FUNCTION_BLOCK PUBLIC FB_BANNER_K50
VAR_IN_OUT
	Hardware : TYP_BAN_K50_HW;
END_VAR
VAR_INPUT
END_VAR
VAR_OUTPUT
	ButtonPressed : BOOL;
	ButtonPosEdge : BOOL;
	ButtonNegEdge : BOOL;
END_VAR
VAR
	PosTrig : R_TRIG;
	NegTrig : F_TRIG;
END_VAR

ButtonPressed := Hardware.In.ButtonPressed;

PosTrig(CLK := ButtonPressed, Q => ButtonPosEdge);
NegTrig(CLK := ButtonPressed, Q => ButtonNegEdge);

METHOD PUBLIC SetGreenLight : REFERENCE TO FB_BANNER_K50
VAR_INPUT
END_VAR
{warning disable C0371}

// Checking the VAR_IN_OUT reference, leave the current method in case of invalid reference
IF NOT __ISVALIDREF(THIS^.Hardware) THEN
     RETURN;
END_IF

THIS^.Hardware.Out.Green := TRUE;

SetGreenLight REF= THIS^;
END_METHOD

METHOD PUBLIC SetRedLight : REFERENCE TO FB_BANNER_K50
VAR_INPUT
END_VAR
{warning disable C0371}

// Checking the VAR_IN_OUT reference, leave the current method in case of invalid reference
IF NOT __ISVALIDREF(THIS^.Hardware) THEN
     RETURN;
END_IF


THIS^.Hardware.Out.Red := TRUE;

SetRedLight REF= THIS^;
END_METHOD

METHOD PUBLIC SetYellowLight : REFERENCE TO FB_BANNER_K50
VAR_INPUT
END_VAR
{warning disable C0371}

// Checking the VAR_IN_OUT reference, leave the current method in case of invalid reference
IF NOT __ISVALIDREF(THIS^.Hardware) THEN
     RETURN;
END_IF


THIS^.Hardware.Out.Yellow := TRUE;

SetYellowLight REF= THIS^;
END_METHOD

METHOD PUBLIC TurnOffLights : REFERENCE TO FB_BANNER_K50
VAR_INPUT
END_VAR
{warning disable C0371}

// Checking the VAR_IN_OUT reference, leave the current method in case of invalid reference
IF NOT __ISVALIDREF(THIS^.Hardware) THEN
     RETURN;
END_IF


THIS^.Hardware.Out.Green := FALSE;
THIS^.Hardware.Out.Yellow := FALSE;
THIS^.Hardware.Out.Red := FALSE;

TurnOffLights REF= THIS^;
END_METHOD

END_FUNCTION_BLOCK

(* stored: Version 1.1.0.1, ProductVersion 3.1.4024.12
   POU FB_BANNER_K50: Id {b592f749-083e-4cee-a196-8c700fdcbac2}, SpecialFunc None
   Method SetGreenLight: Id {7cdfc9b8-e08c-445e-bf0e-fd5eaa830e18}
   Method SetRedLight: Id {ed435eff-65b3-4b2f-bfed-bf5eaa32a982}
   Method SetYellowLight: Id {c1222960-600c-44b0-be57-c6fe1f5ad668}
   Method TurnOffLights: Id {e3bb478d-b2d0-46c4-85ce-bc36ab8e5820} *)
